// TwinCAT 3 PLC project SPS
// ProgramVersion: 3.1.4024.0
// libraries:
//   Tc2_MC2, * (Beckhoff Automation GmbH)
//   Tc2_Standard, * (Beckhoff Automation GmbH)
//   Tc2_System, * (Beckhoff Automation GmbH)
//   Tc3_Module, * (Beckhoff Automation GmbH)
// project tree:
//   DUTs/ eBetriebszustand.TcDUT
//   GVLs/ IFC_HW.TcGVL (not stored)
//   / PlcTask.TcTTO
//   POUs/Ampel/ FB_Ampel.TcPOU, FB_Blinken_Ampel.TcPOU
//   POUs/ FB_EZylinder.TcPOU, FB_Vereinzelung.TcPOU, MAIN.TcPOU
//   POUs/Transport/ FB_Lieferband.TcPOU, FB_Transport.TcPOU, FB_TransportA.TcPOU, FB_TransportE.TcPOU, FB_TransportLogik.TcPOU
// real-time tasks:
//   TASK PlcTask: cycle T#10ms, priority 20, ADS port 350
// motion (NC):
//   TASK NC-Task 1 SAF: cycle T#2ms, priority 4, ADS port 501
//   TASK NC-Task 1 SVB: cycle T#10ms, priority 8, ADS port 511
//   AXIS Achse_Band (id 1)
//     OtherSettings: AllowMotionCmdToSlave=true
//     encoder EncType=1
//     drive DrvType=5
//       Analog: TorqueSetpointScale=10, ScaleFactorActTorque=0.1
//       TimeComp: TaskDelayCycles=1
//     controller CtrType=1
//       CtrPara: PriorControlFactor=1
//         Observer: BandWidth=20
// variable links:
//   SPS/SPS Instance <-> NC-Task 1 SAF/Axes/Achse_Band
//     PlcTask Inputs/IFC_HW.ax_BandMotor.NcToPlc <-> Outputs/ToPlc
//     PlcTask Outputs/IFC_HW.ax_BandMotor.PlcToNc <-> Inputs/FromPlc

CONFIGURATION SPS
    RESOURCE PLC ON TwinCAT3
        TASK PlcTask(INTERVAL := T#10ms, PRIORITY := 20);
        PROGRAM MAIN WITH PlcTask : MAIN;
    END_RESOURCE
END_CONFIGURATION

// ---- DUTs/eBetriebszustand.TcDUT
{attribute 'qualified_only'}
{attribute 'strict'}
TYPE eBetriebszustand :
(
	Off,		//nicht Betriebsbereit						nichts
	Error,		//Fehlerbehafteter Stopp					Gelb -> Blinkt
	Setup,		//Wartung									Rot, Gelb, Grün -> leuchtet
	Warning,	//Nicht Fehlerbehafteter Stopp				Rot -> Blinkt
	Init,		//herstellung Betriebsbereitschaft			Gelb -> leuchtet
	Ready,		//Betriebsbereit							Grün und Gelb -> Blinkt
	Production,	//Betrieb									Grün -> leuchtet
	Done,		//Betrieb abgeschlossen						Grün -> Blinkt
	Stop		//geplanter Stop							Yellow -> leuchtet
);
END_TYPE

// ---- POUs/MAIN.TcPOU
PROGRAM MAIN
VAR
	fbVereinzelung : FB_Vereinzelung;
	fbEZylinder1 : FB_EZylinder;
	fbEZylinder2 : FB_EZylinder;
	
	fbAmpel : FB_Ampel;
	eState: eBetriebszustand;
	
	MCPower : MC_Power;
	
	fbForderband : FB_Lieferband;
	
	fbTransport : FB_Transport;
END_VAR


fbAmpel(eState:= eState, bRed=>IFC_HW.bAmpelRot , bYellow=>IFC_HW.bAmpelGelb , bGreen=>IFC_HW.bAmpelGrun );

IFC_HW.ax_BandMotor.ReadStatus();

MCPower(
	Axis:= IFC_HW.ax_BandMotor, 
	Enable:= TRUE, 
	Enable_Positive:= TRUE, 
	Enable_Negative:= TRUE, 
	Override:= , 
	BufferMode:= , 
	Options:= , 
	Status=> , 
	Busy=> , 
	Error=> , 
	ErrorID=> );


fbVereinzelung(
	bEnable:= IFC_HW.bEnable, 
	bExecute:= IFC_HW.bExecute, 
	bSensor1:= IFC_HW.bEinzelSens1, 
	bSensor2:= IFC_HW.bEinzelSens2, 
	bSensor3:= IFC_HW.bEinzelSens3, 
	bSensor4:= IFC_HW.bBandSens1, 
	bGate1=> fbEZylinder1.bGate, 
	bGate2=> fbEZylinder2.bGate,
	eState=> eState);
	
	
fbEZylinder1(bGate:= , bError:= , bR1=> IFC_HW.bR1AKT1, bR2=> IFC_HW.bR2AKT1);
fbEZylinder2(bGate:= , bError:= , bR1=> IFC_HW.bR1AKT2, bR2=> IFC_HW.bR2AKT2);

fbForderband(
	bEnable:= IFC_HW.bEnable, 
	bExecute:= IFC_HW.bExecute, 
	bHalt:= IFC_HW.bBandSens1, 
	eState=> , 
	ax:= IFC_HW.ax_BandMotor);


(*fbTransport(
	bEnable:=IFC_HW.bEnable, 
	bExecute:= IFC_HW.bExecute, 
	nStation:= , 
	bSens1:= IFC_HW.bBandSens1, 
	bSens2:= IFC_HW.bBandSens2, 
	bSens3:= IFC_HW.bBandSens3, 
	bSens4:= IFC_HW.bBandSens4, 
	eState=> , 
	bStopper1=> IFC_HW.bBandHub1, 
	bStopper2=> IFC_HW.bBandHub2, 
	bStopper3=> IFC_HW.bBandHub3, 
	ax:= IFC_HW.ax_BandMotor); *)

END_PROGRAM

// ---- POUs/FB_Vereinzelung.TcPOU
FUNCTION_BLOCK FB_Vereinzelung
VAR_INPUT
	//Steuervariablen
	bEnable : BOOL;
	bExecute : BOOL;
	//Hardware Eingänge
	bSensor1 : BOOL; //Flasche in der Kammer
	bSensor2 : BOOL; //Flasche im Rohr
	bSensor3 : BOOL; //Flasche auf Kopf
	bSensor4 : BOOL; //Flasche am Förderband
END_VAR
VAR_OUTPUT
	//Hardware Ausgänge
	bGate1: BOOL;
	bGate2: BOOL;
	eState: eBetriebszustand;	
END_VAR
VAR
	nState: INT := 100;

	fbTon: Ton;
END_VAR

fbTon(IN:= , PT:= T#1S, Q=> , ET=> );

CASE nState OF
	100:
	eState := eBetriebszustand.Off;
	
	IF bSensor1 AND bEnable THEN
		nState := 21; //Ready
	ELSIF bEnable THEN
		nState := 0; //Init
	END_IF
	
	0: //Kammer ist leer
	eState := eBetriebszustand.Init;
	bGate1 := FALSE;
	bGate2 := FALSE;
	
	IF bSensor2 THEN
		nState := 1; //Oben öffnen
	END_IF
	
	1: //Oben öffnen
	eState := eBetriebszustand.Init;
	bGate1 := TRUE;
	bGate2 := FALSE;
	
	IF bSensor1 THEN
		nState := 2; //oben schließen
	END_IF
	
	2: //oben schließen
	
	eState := eBetriebszustand.Init;
	bGate1 := FALSE;
	bGate2 := FALSE;
	fbTon.IN := TRUE;
	
	IF bSensor1 THEN
		nState := 21; //Ready
		fbTon.IN := FALSE;
	END_IF
	
	21: //Ready
	eState := eBetriebszustand.Ready;
	bGate1 := FALSE;
	bGate2 := FALSE;
	fbTon.IN := TRUE;
	
	IF bExecute THEN
		nState := 3;
	END_IF
	
	3:	//unten öffen
	eState := eBetriebszustand.Production;
		bGate1 := FALSE;
		bGate2 := TRUE;
		IF bSensor4 THEN
			nState := 4;
		END_IF
	
	4:	//unten schließen
		eState := eBetriebszustand.Production;
		bGate1 := FALSE;
		bGate2 := FALSE;
		IF fbTon.Q THEN
			nState := 41;
		END_IF
	
	41:	//Ablauf fertig
	eState := eBetriebszustand.Done;
		IF NOT bExecute THEN
			nState := 0;
		END_IF
	
	
END_CASE

END_FUNCTION_BLOCK

// ---- POUs/FB_EZylinder.TcPOU
FUNCTION_BLOCK FB_EZylinder
VAR_INPUT
	bGate : BOOL;
	bError : BOOL;
END_VAR
VAR_OUTPUT
	bR1 : BOOL;
	bR2 : BOOL;
END_VAR
VAR
END_VAR


bR1 := bGate;
bR2 := NOT bGate;

IF bError THEN
	bR1 := FALSE;
	bR2 := FALSE;
END_IF

END_FUNCTION_BLOCK

// ---- POUs/Ampel/FB_Ampel.TcPOU
FUNCTION_BLOCK FB_Ampel
VAR_INPUT
	eState : eBetriebszustand;
END_VAR

VAR_OUTPUT
	bRed : BOOL := FALSE;
	bYellow : BOOL := FALSE;
	bGreen : BOOL := FALSE;
END_VAR

VAR
	nState : INT := 0;
	fbTon : Ton;
	fbBlink : FB_Blinken_Ampel;
	bBlinken: BOOL;
END_VAR

CASE nState OF
	
	//Off -> nicht Betriebsbereit
	0: 
		IF eState = eBetriebszustand.Init THEN
			nState := 10;
		END_IF
		
	//Init -> herstellung Betriebsbereitschaft
	10: 
		bYellow := TRUE;
		IF eState = eBetriebszustand.Ready THEN
			bYellow := FALSE;
			nState := 20;
		END_IF
	
	//Ready -> Betriebsbereit
	20:
		fbBlink(tPeriode:= T#1S , bBlink=> bBlinken);
		bGreen := bBlinken;
		bYellow := bBlinken;
		
		IF eState = eBetriebszustand.Production THEN
			bGreen := FALSE;
			bYellow := FALSE;
			nState := 30;
		END_IF
	
	//Production -> Betrieb	
	30: 
		bGreen := TRUE;
		IF eState = eBetriebszustand.Done THEN
			bGreen := FALSE;
			nState := 40;
		END_IF
		
	40: //Done -> Betrieb abgeschlossen
		fbBlink(tPeriode:= T#1S , bBlink=> bBlinken);
		bGreen := bBlinken;
		
	50: //Stop -> geplanter Stop
		bYellow := TRUE;
		
	60: //Setup -> Wartung
		bRed := TRUE;
		bYellow := TRUE;
		bGreen := TRUE;
		
	90://Error -> Fehlerbehafteter Stopp
		fbBlink(tPeriode:= T#1S , bBlink=> bBlinken);
		bYellow := bBlinken;
		
	99: //Warning -> Nicht Fehlerbehafteter Stopp
		fbBlink(tPeriode:= T#1S , bBlink=> bBlinken);
		bRed := bBlinken;
	
END_CASE

END_FUNCTION_BLOCK

// ---- POUs/Ampel/FB_Blinken_Ampel.TcPOU
FUNCTION_BLOCK FB_Blinken_Ampel
VAR_INPUT
	tPeriode  : TIME := T#1S;   // Gesamtperiode des Blinkens
END_VAR
VAR_OUTPUT
	bBlink : BOOL := FALSE;     // Ausgang: Blinkt true/false
END_VAR
VAR
	fbTon : TON;                // Einschalt-Timer
END_VAR

// Timer läuft dauerhaft
fbTon(IN := TRUE, PT := tPeriode);

// Blink-Logik: 50/50 Duty Cycle
IF fbTon.ET < tPeriode / 2 THEN
	bBlink := TRUE;
ELSE
	bBlink := FALSE;
END_IF

// Timer neu starten, wenn abgelaufen
IF fbTon.Q THEN
	fbTon(IN := FALSE);  // kurzer Reset
END_IF

END_FUNCTION_BLOCK

// ---- POUs/Transport/FB_Lieferband.TcPOU
FUNCTION_BLOCK FB_Lieferband
VAR_INPUT
	//Steuereingänge
	bEnable : BOOL;
	bExecute : BOOL;
	bHalt : BOOL;
END_VAR
VAR_OUTPUT
	eState : eBetriebszustand;
END_VAR
VAR
	nState : INT := 0;
	rVelocity : REAL;
	rAcceleration : REAL;
	// Motion Blöcke der Tc2_Mc2
	mcReset : MC_Reset;
	mcPower : MC_Power;
	mcVelocity : MC_MoveVelocity;
	mcHalt : MC_Halt;
END_VAR

VAR_IN_OUT
	ax : Axis_Ref;
END_VAR

ax.ReadStatus(); //Aktualisierung der Position für das Förderband in der Teaching Factory 
//Ausschreiben des Funktionsbausteines 
mcReset(
	Axis:= ax,  
	Execute:= , 
	Done=> , 
	Busy=> , 
	Error=> , 
	ErrorID=> );
	
mcPower(
	Axis:= ax, //Weitere Parameter über Punkt-Notation 
	Enable:= , 
	Enable_Positive:= , 
	Enable_Negative:= , 
	Override:= , 
	BufferMode:= , 
	Options:= , 
	Status=> , 
	Busy=> , 
	Error=> , 
	ErrorID=> );

mcVelocity(
	Axis:= ax, 
	Execute:= , 
	Velocity:= , 
	Acceleration:= , 
	Deceleration:= , 
	Jerk:= , 
	Direction:= MC_Positive_Direction, 
	BufferMode:= , 
	Options:= , 
	InVelocity=> , 
	Busy=> , 
	Active=> , 
	CommandAborted=> , 
	Error=> , 
	ErrorID=> );

mcHalt(
	Axis:= ax, 
	Execute:= , 
	Deceleration:= 60, 
	Jerk:= , 
	BufferMode:= , 
	Options:= , 
	Done=> , 
	Busy=> , 
	Active=> , 
	CommandAborted=> , 
	Error=> , 
	ErrorID=> );
	
//Zustandsdiagramm nach Unterricht

IF NOT mcPower.Status THEN
	nState := 0;
END_IF

CASE nState OF
	0: 
		eState := eBetriebszustand.Off;
		mcPower.Enable := TRUE;
		mcPower.Enable_Positive := TRUE;
		
		IF mcPower.Status AND bEnable THEN
			nState := 20;
		ELSIF bEnable AND NOT mcPower.Status THEN
			nState := 10;
		END_IF
	
	10:
		eState := eBetriebszustand.Init;
		mcReset.Execute := TRUE;
		mcPower.Enable := FALSE;
		IF mcReset.Done THEN
			nState := 11;
		END_IF
	
	11:
		eState := eBetriebszustand.Init;
		mcPower.Enable := TRUE;
		mcReset.Execute := FALSE;
		IF mcPower.Status THEN
			nState := 20;
		END_IF
		
	20:
		eState := eBetriebszustand.Ready;
		IF bExecute THEN
			nState := 30;		
		END_IF
	
	30:
		eState := eBetriebszustand.Production;
		mcVelocity.Execute := TRUE;
		mcVelocity.Velocity := 30;
		mcVelocity.Acceleration := 60;
		IF bHalt THEN
			nState := 31;
		END_IF
	
	31:
		eState := eBetriebszustand.Production;
		mcVelocity.Execute := FALSE;
		mcHalt.Execute := TRUE;
		mcHalt.Deceleration := 60;
		IF mcHalt.Done THEN
			nState := 40;
		END_IF
	
	40:
		eState := eBetriebszustand.Done;
		mcHalt.Execute := FALSE;
		IF NOT bExecute THEN
			nState := 20;
		END_IF
END_CASE

END_FUNCTION_BLOCK

// ---- POUs/Transport/FB_Transport.TcPOU
FUNCTION_BLOCK FB_Transport
VAR_INPUT
	bEnable : BOOL;
	bExecute : BOOL;
	nStation : INT;
	//Hardwdare Eingänge
	bSens1 : BOOL;
	bSens2 : BOOL;
	bSens3 : BOOL;
	bSens4 : BOOL;
END_VAR
VAR_OUTPUT
	eState : eBetriebszustand;
	bStopper1 : BOOL;
	bStopper2 : BOOL;
	bStopper3 : BOOL;
END_VAR
VAR
	fbTransportE : FB_TransportE;
	fbTransportLogik : FB_TransportLogik;
	fbTransportA : FB_TransportA;
	fbLieferband : FB_Lieferband;
END_VAR
VAR_IN_OUT
	//Achsen Ref
	ax : Axis_Ref;
END_VAR

fbTransportE(
	bSens1:= , 
	bSens2:= , 
	bSens3:= , 
	bSens4:= , 
	bStation1=> , 
	bStation2=> , 
	bStation3=> , 
	bStation4=> );
	
fbTransportLogik(
	bEnable:= bEnable , 
	bExecute:= bExecute , 
	eStateE:= fbLieferband.eState, 
	nStation:= nStation, 
	bStation1:= fbTransportE.bStation1, 
	bStation2:= fbTransportE.bStation2, 
	bStation3:= fbTransportE.bStation3, 
	bStation4:= fbTransportE.bStation4, 
	bEnableA=> , 
	bExecuteA=> , 
	bStopA=> , 
	eStateA=> , 
	bStop1=> , 
	bStop2=> , 
	bStop3=> );
	
fbLieferband(
	bEnable:= fbTransportLogik.bEnableA , 
	bExecute:= fbTransportLogik.bExecuteA , 
	bHalt:= fbTransportLogik.bStopA, 
	eState=> , 
	ax:= ax);
	
fbTransportA(
	bStop1:= fbTransportLogik.bStop1, 
	bStop2:= fbTransportLogik.bStop2, 
	bStop3:= fbTransportLogik.bStop3, 
	bStopper1=> bStopper1, 
	bStopper2=> bStopper2, 
	bStopper3=> bStopper3);

END_FUNCTION_BLOCK

// ---- POUs/Transport/FB_TransportE.TcPOU
FUNCTION_BLOCK FB_TransportE
VAR_INPUT
	bSens1 : BOOL;
	bSens2 : BOOL;
	bSens3 : BOOL;
	bSens4 : BOOL;
END_VAR
VAR_OUTPUT
	bStation1 : BOOL;
	bStation2 : BOOL;
	bStation3 : BOOL;
	bStation4 : BOOL;
END_VAR
VAR
END_VAR

bStation1 := bSens1;
bStation2 := bSens2;
bStation3 := bSens3;
bStation4 := bSens4;

END_FUNCTION_BLOCK

// ---- POUs/Transport/FB_TransportLogik.TcPOU
FUNCTION_BLOCK FB_TransportLogik
VAR_INPUT
	bEnable : BOOL;
	bExecute : BOOL;
	eStateE : eBetriebszustand;
	nStation : INT;
	// Logik -> Hardware Signal
	bStation1 : BOOL;
	bStation2 : BOOL;
	bStation3 : BOOL;
	bStation4 : BOOL;
END_VAR
VAR_OUTPUT
	bEnableA : BOOL;
	bExecuteA : BOOL;
	bStopA : BOOL;
	eStateA: eBetriebszustand;
	bStop1 : BOOL;
	bStop2 : BOOL;
	bStop3 : BOOL;
END_VAR
VAR
	nState : INT;
END_VAR

END_FUNCTION_BLOCK

// ---- POUs/Transport/FB_TransportA.TcPOU
FUNCTION_BLOCK FB_TransportA
VAR_INPUT
	bStop1 : BOOL;
	bStop2 : BOOL;
	bStop3 : BOOL;
END_VAR
VAR_OUTPUT
	bStopper1 : BOOL;
	bStopper2 : BOOL;
	bStopper3 : BOOL;
END_VAR
VAR
END_VAR

bStopper1 := bStop1;
bStopper2 := bStop2;
bStopper3 := bStop3;

END_FUNCTION_BLOCK
